// TwinCAT 3 PLC project Untitled1
// ProgramVersion: 3.1.4024.12
// libraries:
//   Tc2_Standard, * (Beckhoff Automation GmbH)
//   Tc2_System, * (Beckhoff Automation GmbH)
//   Tc2_Utilities, * (Beckhoff Automation GmbH)
//   Tc3_EventLogger, * (Beckhoff Automation GmbH)
//   Tc3_Module, * (Beckhoff Automation GmbH)
// project tree:
//   GVLs/ HMI.TcGVL
//   / PlcTask.TcTTO
//   POUs/Alarm/ Alarm.TcPOU, FB_ExportCSV.TcPOU
//   POUs/ MAIN.TcPOU
// real-time tasks:
//   TASK PlcTask: cycle T#10ms, priority 20, ADS port 350

CONFIGURATION Untitled1
    RESOURCE PLC ON TwinCAT3
        TASK PlcTask(INTERVAL := T#10ms, PRIORITY := 20);
        PROGRAM MAIN WITH PlcTask : MAIN;
    END_RESOURCE
END_CONFIGURATION

// ---- GVLs/HMI.TcGVL
{attribute 'qualified_only'}
VAR_GLOBAL
	clearAlarmAll : BOOL;
	bExportCSV : BOOL;
	clearlogged : BOOL;
	AlarmID: UINT;
END_VAR

// ---- POUs/MAIN.TcPOU
PROGRAM MAIN
VAR
	al : Alarm;
	a2 : Alarm;
	
	raise: BOOL;
	confirm : BOOL;
	clear : BOOL;
	
	raise2: BOOL;
	confirm2 : BOOL;
	clear2 : BOOL;
	
	clearAlarms : BOOL; 
	fbEventLogger : FB_TcEventLogger;
	iEventLoggerSetting : I_TcClearLoggedEventsSettings;
	fbEventLoggerSetting : FB_TcClearLoggedEventsSettings;
END_VAR

al(
	AlarmID := TC_Events.Alarm.Event,
	bRaiseAlarm := raise);

a2(
	AlarmID := TC_Events.Alarm.AlarmEvent2,
	bRaiseAlarm := raise2);
clearAlarms := HMI.clearAlarmAll;	
FB_ExportCSV(bExport := HMI.bExportCSV);
ClearLoggedEvent(HMI.clearlogged);

METHOD ClearLoggedEvent : BOOL
VAR_INPUT
	bClearLoggedEvent : BOOL;
END_VAR

VAR
	
	clear : BOOL;
END_VAR
IF bClearLoggedEvent THEN
	fbEventLoggerSetting.Clear();
	//fbEventLogger.ClearAllAlarms(0, bClearLoggedEvent);	
	fbEventLogger.ConfirmAllAlarms(0);
	clearAlarms := TRUE;
	FB_ExportCSV(bExport := TRUE);	
	fbEventLogger.ClearLoggedEvents(fbEventLoggerSetting);
	bClearLoggedEvent := FALSE;
	
END_IF
END_METHOD

END_PROGRAM

// ---- POUs/Alarm/Alarm.TcPOU
FUNCTION_BLOCK Alarm
VAR_INPUT
	AlarmID : TcEventEntry;
	bRaiseAlarm : BOOL :=0;
	bConfirmAlarm : BOOL := 0;
    bClearAlarm : BOOL := 0;
	
END_VAR
VAR_OUTPUT
END_VAR
VAR
	
	bRaise : BOOL :=0;	
	bIsInitalized : BOOL :=0;
	nTimeStamp : ULINT := 0;
	fbAlarm : FB_TcALarm;
	
END_VAR

Initalize();
RaiseAlarm();
ConfirmAlarm();
ClearAlarm();
//ClearLoggedEvent();

METHOD ClearAlarm : BOOL
VAR
	bClearALL : BOOL;
END_VAR
bclearALL := MAIN.clearAlarms;
IF NOT bRaiseAlarm THEN //
	IF bClearAlarm OR bClearALL THEN	
		fbAlarm.Clear(nTimeStamp, FALSE);
	END_IF
END_IF
END_METHOD

METHOD ConfirmAlarm : BOOL
VAR_INPUT
END_VAR
IF bConfirmAlarm THEN
	fbAlarm.Confirm(nTimeStamp);
END_IF
END_METHOD

METHOD Initalize : BOOL
VAR
	fbSourceInfo : FB_TcSourceInfo;
END_VAR
IF NOT bIsInitalized THEN
	bIsInitalized := TRUE;
	//fbSourceInfo.sName := UDINT_TO_STRING(AlarmID.nEventId);
	fbAlarm.CreateEx(AlarmID, TRUE, fbSourceInfo);
END_IF
END_METHOD

METHOD RaiseAlarm : BOOL
VAR

END_VAR
bRaise := bRaiseAlarm;
IF bRaise THEN
	fbAlarm.Raise(nTimeStamp);
END_IF
END_METHOD

END_FUNCTION_BLOCK

// ---- POUs/Alarm/FB_ExportCSV.TcPOU
PROGRAM FB_ExportCSV
VAR_INPUT
	bExport				: BOOL;
END_VAR

VAR
	hr : HRESULT;
	
	fbCsvExportSetting	: FB_TcEventCsvExportSettings; 
	fbExportFilter		: I_TcEventFilter; 
	sExportFilePath		: T_maxString := 'C:\dataCollection\';
	sExportFileName		: T_maxString := 'Alarms_History.csv';
	
	fbEventLogger	: FB_TcEventLogger;
	fbTrig			: R_TRIG;
	
	getTime : FB_LocalSystemTime := ( bEnable := TRUE, dwCycle := 5 );
	dateStr : T_MaxString;
END_VAR

getTime();
fbTrig(CLK:=bExport);
IF bExport THEN
	IF fbTrig.Q THEN 
		dateStr := getDateStr();
		sExportFileName	:= Concat(Concat(sExportFilePath,'Alarms_History_'),Concat(dateStr,'.csv'));
		fbCsvExportSetting.Clear();
		fbCsvExportSetting.sDelimiter := ',' ;
		//fbCsvExportSetting.AddLanguage(1031, 'German');
		fbCsvExportSetting.AddFilter(fbExportFilter); 
		//fbExportFilter.Clear().IsMessage().AND_OP().EventClass.EqualTo(TC_EVENTS.Alarm.Event.uuidEventClass);
	END_IF
	IF fbEventLogger.ExportLoggedEvents(sExportFileName, fbCsvExportSetting, hrErrorCode=>hr) THEN // async request returns TRUE if not any more busy 
		bExport := FALSE;
	END_IF
END_IF

METHOD getDateStr : T_MaxString
VAR_INPUT
END_VAR
getDateStr := CONCAT(WORD_TO_STRING(getTime.systemTime.wMonth), CONCAT('_', CONCAT(WORD_TO_STRING(getTime.systemTime.wDay), CONCAT('_', WORD_TO_STRING(getTime.systemTime.wYear)))));
END_METHOD

END_PROGRAM
